// TIA Portal V19 export
TYPE "Thickness_Measure_Item"
   STRUCT
      ID : DInt;   // Measure ID
      Time_Stamp : DTL;   // Time stamp
      Status : Int;   // 0=NULL; 1=OK; 2=NG
      Material_Position : LReal;   // Material Position where the Reading was done
      Value : Real;   // Sensore value
      Err : Real;   // Sensor deviation from target value
      Avg : Real;   // Average value
      AvgErr : Real;   // Average value deviation from target value
   END_STRUCT;
END_TYPE
